// TIA Portal V17 export
// export: Created 2023-04-19T10:28:58.0904628Z, ExportSetting WithDefaults, DisplayName Totally Integrated Automation Portal, DisplayVersion V17, DisplayName TIA Portal Openness, DisplayVersion V17, DisplayName TIA Portal Version Control Interface, DisplayVersion V17, DisplayName STEP 7 Professional, DisplayVersion V17, DisplayName STEP 7 Safety, DisplayVersion V17, DisplayName WinCC Advanced, DisplayVersion V17
DATA_BLOCK "FB_Testblok_DB"   // DB1
VERSION : 0.1
// stored: AutoNumber true, DBAccessibleFromOPCUA true, InstanceOfName FB_Testblok, InstanceOfType FB
"FB_Testblok"
   // VAR_INPUT
   //    Input_Int : Int;
   // END_VAR
   // VAR_OUTPUT
   //    Output_Real : Real;
   // END_VAR
BEGIN
END_DATA_BLOCK
